Staubli VAL3: IO.pgx

program IO()
begin

  //Read and process external controller information
  while bError==false

    nStart=clock()
    nDelay = clock()-nStart

    bEstAtornillador=dDioEstAtornillador
    bEstPinza=dDioEstPinza
    bHerramientaRobot=dDioHerramientaRobot
    bTLocked=dDioTLocked
    bTUnlocked=dDioTUnlocked
    dDioMoveGripper=bMoveGripper


    if dESbutton == true
      dDioEmergencyButton = true
    else
      dDioEmergencyButton = false
    endIf

    if dDoor1 == true
      dDioDoor1Status = true
    else
      dDioDoor1Status = false
    endIf

    if dDoor2 == true
      dDioDoor2Status = true
    else
      dDioDoor2Status = false
    endIf

    delay(0)
  endWhile

end
